// TIA Portal V16 export
// export: Created 2021-07-12T14:47:16.8522022Z, ExportSetting WithDefaults, DisplayName Totally Integrated Automation Portal, DisplayVersion V16, DisplayName TIA Portal Version Control Interface, DisplayVersion V16, DisplayName TIA Portal Openness, DisplayVersion V16, DisplayName STEP 7 Professional, DisplayVersion V16, DisplayName STEP 7 Safety, DisplayVersion V16, DisplayName WinCC Professional, DisplayVersion V16
DATA_BLOCK "SimaHydTO_AdvancedAxisControl_DB"   // DB4
FAMILY : SimaHydTO
VERSION : 1.0
// stored: AutoNumber true, DBAccessibleFromOPCUA true, InstanceOfName SimaHydTO_AdvancedAxisControl, InstanceOfType FB
"SimaHydTO_AdvancedAxisControl"
   // VAR_IN_OUT
   //    hmiConnection : "SimaHydTO_typeHMIConnection";
   //    axisData : "LSimaHydTO_typeAxisData";
   //    axesArray : Array[*] of "SimaHydTO_typeAxesArray";
   // END_VAR
   // VAR
   //    statActualAxisIndex { ExternalAccessible := 'False'; ExternalVisible := 'False'; ExternalWritable := 'False'} : Int;
   //    statAxisIndexOld { ExternalAccessible := 'False'; ExternalVisible := 'False'; ExternalWritable := 'False'} : Int;
   //    instSimaHydTO_AxisAdvancedPosAxis { ExternalAccessible := 'False'; ExternalVisible := 'False'; ExternalWritable := 'False'; S7_SetPoint := 'True'} : "SimaHydTO_AxisAdvanced_PosAxis";
   //    instSimaHydTO_AxisAdvancedSyncAxis { ExternalAccessible := 'False'; ExternalVisible := 'False'; ExternalWritable := 'False'; S7_SetPoint := 'True'} : "SimaHydTO_AxisAdvanced_SyncAxis";
   // END_VAR
BEGIN
END_DATA_BLOCK
